TYPE (* The class name for generic types *)
  (* Standard: 61499-1; Description: Copyright (c) 2024 Martin Erich Jobst This program and the accompanying materials are made available under the terms of the Eclipse Public License 2.0 which is available at https://www.eclipse.org/legal/epl-2.0/ SPDX-License-Identifier: EPL-2.0 *)
  (* Version 1.0, 2024-08-21, Martin Erich Jobst, initial API and implementation and/or initial documentation *)
  {SET_ATTRIBUTE(TARGET, (IInterfaceElement:=FALSE,SubApp:=FALSE,FBType:=TRUE,Application:=FALSE,Connection:=FALSE,FB:=FALSE,DataType:=FALSE))}
  GenericClassName : STRING := 'GEN_'; (* The class name for generic types *)
END_TYPE
